PROGRAM MAIN
VAR
END_VAR

//prg_KantoorVerlichting();
//prg_Thermostaatregeling();
prg_ThermostaatregelingTijdsturing();

END_PROGRAM

(* stored: Version 1.1.0.1, ProductVersion 3.1.4024.15
   POU MAIN: Id {4131371c-dfa1-4455-b08e-997c10203188}, SpecialFunc None *)
